TYPE DUT_ModelInfo :
STRUCT
	sName		: STRING;
	abType		: ARRAY[0..cMaxTypeNo-1] OF BOOL;
	aiType		: ARRAY[0..cMaxTypeNo-1] OF INT;
	arPosition	: ARRAY[0..cMaxAxisNo-1] OF LREAL;
	arSpeed		: ARRAY[0..cMaxAxisNo-1] OF LREAL;
END_STRUCT
END_TYPE

(* stored: Version 1.1.0.1
   DUT DUT_ModelInfo: Id {e045def9-7134-4c9c-a39f-98f9b517554b} *)
